// TIA Portal project "FactoryIO_assembler_analog" (V19)
// Vorlageprojekt für das Buch mit Zielsystem S7-1200

(* hardware
DEVICE "S7-1200-Station_1"  S7-1200 Station
   slot 0: "Baugruppenträger_0"  Rack  V1.0
   slot 1: "PLC_1"  CPU 1211C DC/DC/DC  6ES7 211-1AE40-0XB0  V4.1
*)

// ===== PLC "PLC_1"  CPU 1211C DC/DC/DC =====

VAR_GLOBAL   // PLC tag table "Standard-Variablentabelle"
   "lids_conveyor1" AT %A0.0 : Bool;
   "item_detected" AT %E0.0 : Bool;
   "lid_at_place" AT %E0.1 : Bool;
   "base_at_place" AT %I0.2 : Bool;
   "part_leaving" AT %I0.3 : Bool;
   "start" AT %I0.4 : Bool;
   "reset" AT %I0.5 : Bool;
   "stop" AT %I0.6 : Bool;
   "emergency_stop" AT %I0.7 : Bool;
   "auto" AT %I1.0 : Bool;
   "game_reset" AT %I1.1 : Bool;
   "x" AT %ID30 : Real;
   "z" AT %ID34 : Real;
   "stop_blade1" AT %Q0.1 : Bool;
   "lids_conveyor2" AT %Q0.2 : Bool;
   "bases_conveyor1" AT %Q0.3 : Bool;
   "stop_blade2" AT %Q0.4 : Bool;
   "bases_conveyor2" AT %Q0.5 : Bool;
   "grab" AT %Q0.6 : Bool;
   "start_light" AT %Q0.7 : Bool;
   "reset_light" AT %Q1.0 : Bool;
   "stop_light" AT %Q1.1 : Bool;
   "set_x" AT %QD30 : Real;
   "set_z" AT %QD34 : Real;
   "Counter" AT %QD38 : DInt;
   "Tag_1" AT %M0.0 : Bool;
   "Tag_2" AT %M0.1 : Bool;
   "Tag_3" AT %M0.2 : Bool;
   "item_detected_bit" AT %M0.3 : Bool;
   "grab_bit" AT %M0.4 : Bool;
   "pick_complete_bit" AT %M0.5 : Bool;
   "place_complete_bit" AT %M0.6 : Bool;
   "is_reset" AT %M0.7 : Bool;
   "home_complete_bit" AT %M1.0 : Bool;
   "Tag_4" AT %M1.1 : Bool;
END_VAR

FUNCTION "conveyor" : Void   // FC1, LAD
{ S7_Optimized_Access := 'TRUE' }
VERSION : 0.1
   VAR_TEMP   // added for the SCL form of the ladder/FBD networks
      _w1 : Bool;
      _w2 : Bool;
   END_VAR
BEGIN

REGION Network 1
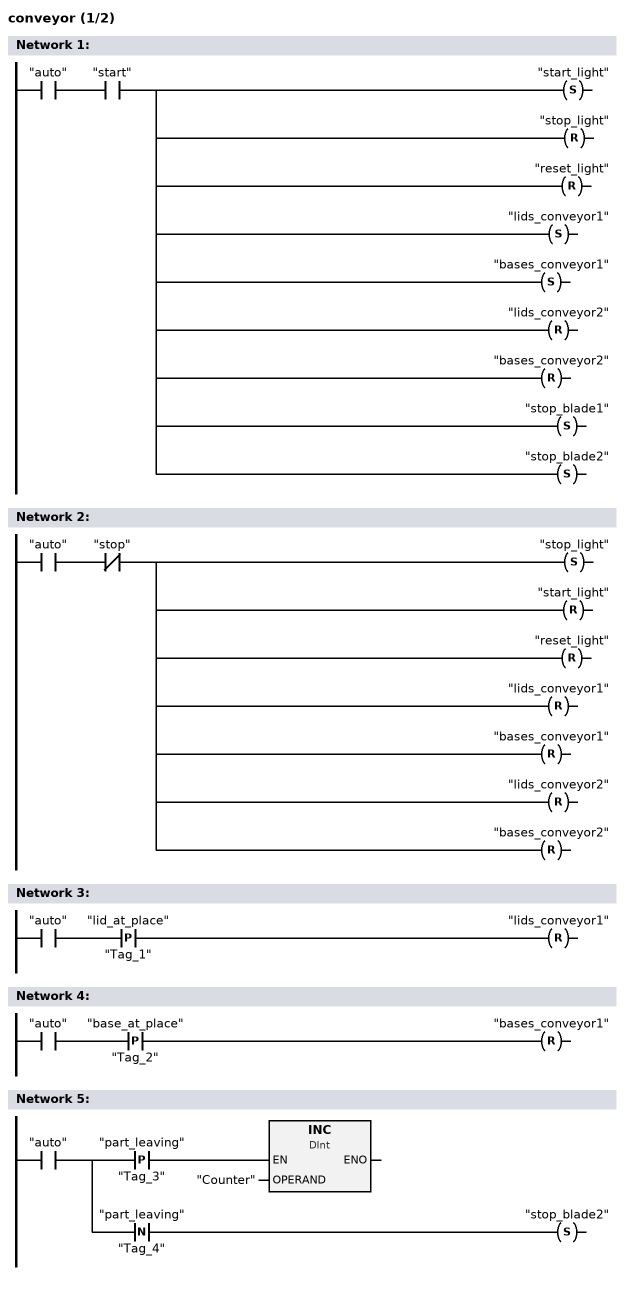
   RUNG wire#powerrail
      Contact( "auto" )
      Contact( "start" )
      wire#w1
      S_Coil( "start_light" )
   END_RUNG
   RUNG wire#w1
      R_Coil( "stop_light" )
   END_RUNG
   RUNG wire#w1
      R_Coil( "reset_light" )
   END_RUNG
   RUNG wire#w1
      S_Coil( "lids_conveyor1" )
   END_RUNG
   RUNG wire#w1
      S_Coil( "bases_conveyor1" )
   END_RUNG
   RUNG wire#w1
      R_Coil( "lids_conveyor2" )
   END_RUNG
   RUNG wire#w1
      R_Coil( "bases_conveyor2" )
   END_RUNG
   RUNG wire#w1
      S_Coil( "stop_blade1" )
   END_RUNG
   RUNG wire#w1
      S_Coil( "stop_blade2" )
   END_RUNG
   // the same network as SCL:
   IF "auto" AND "start" THEN
       "start_light" := TRUE;
       "stop_light" := FALSE;
       "reset_light" := FALSE;
       "lids_conveyor1" := TRUE;
       "bases_conveyor1" := TRUE;
       "lids_conveyor2" := FALSE;
       "bases_conveyor2" := FALSE;
       "stop_blade1" := TRUE;
       "stop_blade2" := TRUE;
   END_IF;
END_REGION

REGION Network 2
   RUNG wire#powerrail
      Contact( "auto" )
      I_Contact( "stop" )
      wire#w1
      S_Coil( "stop_light" )
   END_RUNG
   RUNG wire#w1
      R_Coil( "start_light" )
   END_RUNG
   RUNG wire#w1
      R_Coil( "reset_light" )
   END_RUNG
   RUNG wire#w1
      R_Coil( "lids_conveyor1" )
   END_RUNG
   RUNG wire#w1
      R_Coil( "bases_conveyor1" )
   END_RUNG
   RUNG wire#w1
      R_Coil( "lids_conveyor2" )
   END_RUNG
   RUNG wire#w1
      R_Coil( "bases_conveyor2" )
   END_RUNG
   // the same network as SCL:
   IF "auto" AND NOT "stop" THEN
       "stop_light" := TRUE;
       "start_light" := FALSE;
       "reset_light" := FALSE;
       "lids_conveyor1" := FALSE;
       "bases_conveyor1" := FALSE;
       "lids_conveyor2" := FALSE;
       "bases_conveyor2" := FALSE;
   END_IF;
END_REGION

REGION Network 3
   RUNG wire#powerrail
      Contact( "auto" )
      P_Contact(operand := "lid_at_place", bit := "Tag_1")
      R_Coil( "lids_conveyor1" )
   END_RUNG
   // the same network as SCL:
   #_w1 := "auto" AND "lid_at_place" AND NOT "Tag_1";   // rising edge of "lid_at_place"
   "Tag_1" := "lid_at_place";
   IF #_w1 THEN "lids_conveyor1" := FALSE; END_IF;
END_REGION

REGION Network 4
   RUNG wire#powerrail
      Contact( "auto" )
      P_Contact(operand := "base_at_place", bit := "Tag_2")
      R_Coil( "bases_conveyor1" )
   END_RUNG
   // the same network as SCL:
   #_w1 := "auto" AND "base_at_place" AND NOT "Tag_2";   // rising edge of "base_at_place"
   "Tag_2" := "base_at_place";
   IF #_w1 THEN "bases_conveyor1" := FALSE; END_IF;
END_REGION

REGION Network 5
   RUNG wire#powerrail
      Contact( "auto" )
      wire#w1
      P_Contact(operand := "part_leaving", bit := "Tag_3")
      { S7_Templates := "DestType := DInt" } Inc( "Counter" )
   END_RUNG
   RUNG wire#w1
      N_Contact(operand := "part_leaving", bit := "Tag_4")
      S_Coil( "stop_blade2" )
   END_RUNG
   // the same network as SCL:
   #_w1 := "auto" AND "part_leaving" AND NOT "Tag_3";   // rising edge of "part_leaving"
   "Tag_3" := "part_leaving";
   IF #_w1 THEN "Counter" := "Counter" + 1; END_IF;
   #_w2 := "auto" AND NOT "part_leaving" AND "Tag_4";   // falling edge of "part_leaving"
   "Tag_4" := "part_leaving";
   IF #_w2 THEN "stop_blade2" := TRUE; END_IF;
END_REGION

REGION Network 6
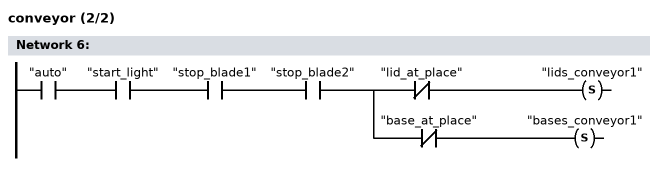
   RUNG wire#powerrail
      Contact( "auto" )
      Contact( "start_light" )
      Contact( "stop_blade1" )
      Contact( "stop_blade2" )
      wire#w1
      I_Contact( "lid_at_place" )
      S_Coil( "lids_conveyor1" )
   END_RUNG
   RUNG wire#w1
      I_Contact( "base_at_place" )
      S_Coil( "bases_conveyor1" )
   END_RUNG
   // the same network as SCL:
   #_w1 := "auto" AND "start_light" AND "stop_blade1" AND "stop_blade2";
   IF #_w1 AND NOT "lid_at_place" THEN "lids_conveyor1" := TRUE; END_IF;
   IF #_w1 AND NOT "base_at_place" THEN "bases_conveyor1" := TRUE; END_IF;
END_REGION
END_FUNCTION

FUNCTION "pick_and_place" : Void   // FC2, LAD
{ S7_Optimized_Access := 'TRUE' }
VERSION : 0.1
   VAR_TEMP
      grab_lid_x_low_limit : Real;
      grab_lid_x_high_limit : Real;
      grab_lid_z_low_limit : Real;
      grab_lid_z_high_limit : Real;
      pick_lid_z_low_limit : Real;
      pick_lid_z_high_limit : Real;
      place_lid_x_low_limit : Real;
      place_lid_x_high_limit : Real;
      place_lid_z_low_limit : Real;
      place_lid_z_high_limit : Real;
   END_VAR
   VAR CONSTANT
      grab_lid_z : Real := 9.3;
      grab_lid_x : Real := 1.2;
      offset : Real := 0.01;
      pick_lid_z : Real;
      place_lid_x : Real := 9.0;
      place_lid_z : Real := 8.95;
      home_z : Real;
      home_x : Real;
   END_VAR
   VAR_TEMP   // added for the SCL form of the ladder/FBD networks
      _w1 : Bool;
      _w2 : Bool;
   END_VAR
BEGIN

REGION Network 1 (SCL)
   // Compute limits
   // 
   #grab_lid_x_high_limit := #grab_lid_x + #offset;
   #grab_lid_x_low_limit := #grab_lid_x - #offset;

   #grab_lid_z_high_limit := #grab_lid_z + #offset;
   #grab_lid_z_low_limit := #grab_lid_z - #offset;

   #pick_lid_z_high_limit := #pick_lid_z + #offset;
   #pick_lid_z_low_limit := MAX(IN1:=0.0, IN2:=#pick_lid_z - #offset);

   #place_lid_x_high_limit:= #place_lid_x + #offset;
   #place_lid_x_low_limit:= #place_lid_x - #offset;

   #place_lid_z_high_limit:= #place_lid_z + #offset;
   #place_lid_z_low_limit:= #place_lid_z - #offset;
END_REGION

REGION Network 2: detect item
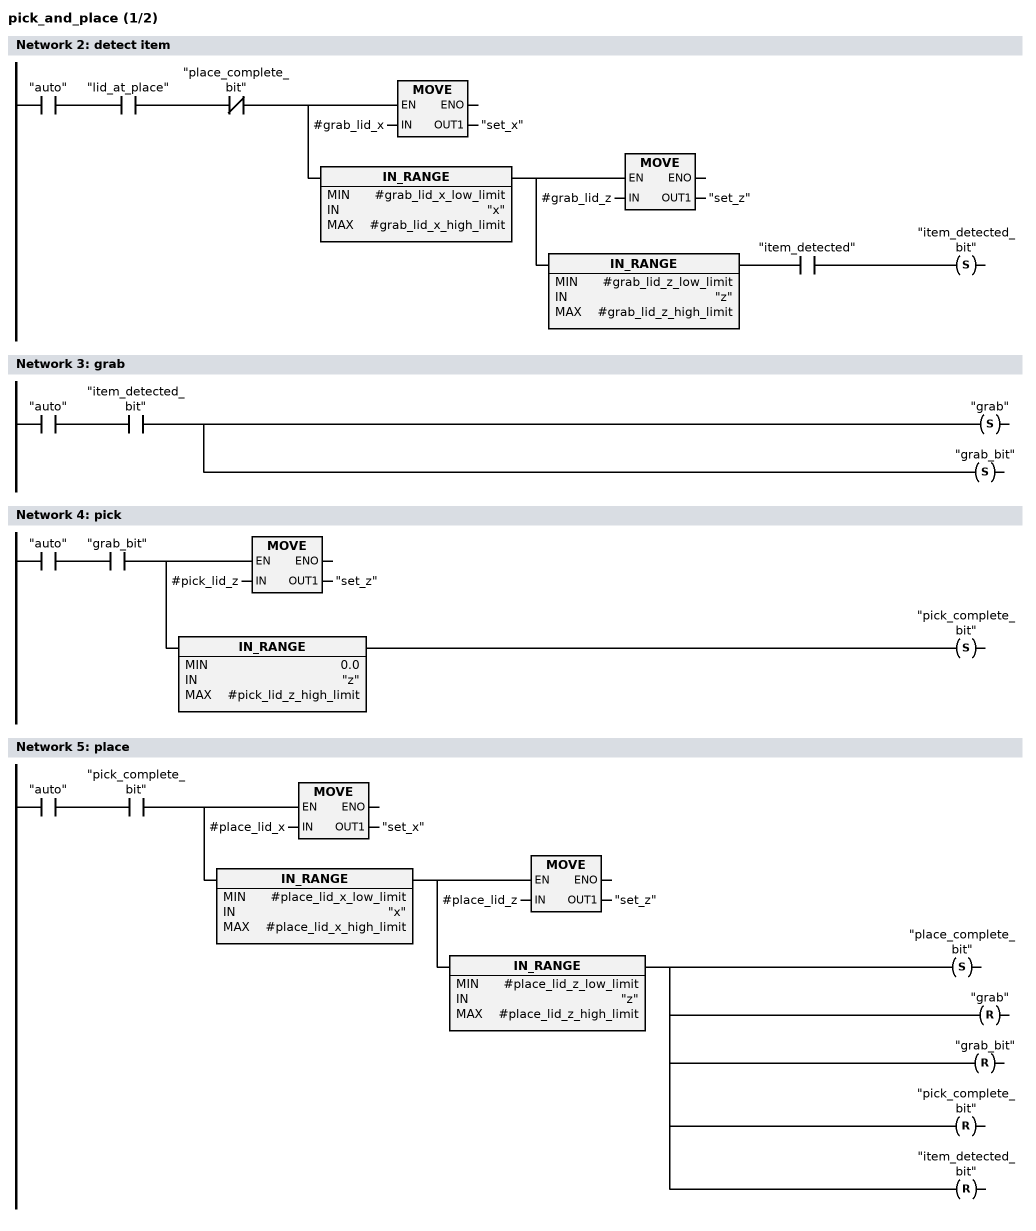
   RUNG wire#powerrail
      Contact( "auto" )
      Contact( "lid_at_place" )
      I_Contact( "place_complete_bit" )
      wire#w1
      Move(in := #grab_lid_x, out1 => "set_x")
   END_RUNG
   RUNG wire#w1
      { S7_Templates := "SrcType := Real" } InRange(min := #grab_lid_x_low_limit, in := "x", max := #grab_lid_x_high_limit)
      wire#w2
      Move(in := #grab_lid_z, out1 => "set_z")
   END_RUNG
   RUNG wire#w2
      { S7_Templates := "SrcType := Real" } InRange(min := #grab_lid_z_low_limit, in := "z", max := #grab_lid_z_high_limit)
      Contact( "item_detected" )
      S_Coil( "item_detected_bit" )
   END_RUNG
   // the same network as SCL:
   #_w1 := "auto" AND "lid_at_place" AND NOT "place_complete_bit";
   IF #_w1 THEN "set_x" := #grab_lid_x; END_IF;
   #_w2 := #_w1 AND (#grab_lid_x_low_limit <= "x") AND ("x" <= #grab_lid_x_high_limit);
   IF #_w2 THEN "set_z" := #grab_lid_z; END_IF;
   IF #_w2 AND (#grab_lid_z_low_limit <= "z") AND ("z" <= #grab_lid_z_high_limit) AND "item_detected" THEN
       "item_detected_bit" := TRUE;
   END_IF;
END_REGION

REGION Network 3: grab
   RUNG wire#powerrail
      Contact( "auto" )
      Contact( "item_detected_bit" )
      wire#w1
      S_Coil( "grab" )
   END_RUNG
   RUNG wire#w1
      S_Coil( "grab_bit" )
   END_RUNG
   // the same network as SCL:
   IF "auto" AND "item_detected_bit" THEN
       "grab" := TRUE;
       "grab_bit" := TRUE;
   END_IF;
END_REGION

REGION Network 4: pick
   RUNG wire#powerrail
      Contact( "auto" )
      Contact( "grab_bit" )
      wire#w1
      Move(in := #pick_lid_z, out1 => "set_z")
   END_RUNG
   RUNG wire#w1
      { S7_Templates := "SrcType := Real" } InRange(min := 0.0, in := "z", max := #pick_lid_z_high_limit)
      S_Coil( "pick_complete_bit" )
   END_RUNG
   // the same network as SCL:
   #_w1 := "auto" AND "grab_bit";
   IF #_w1 THEN "set_z" := #pick_lid_z; END_IF;
   IF #_w1 AND (0.0 <= "z") AND ("z" <= #pick_lid_z_high_limit) THEN "pick_complete_bit" := TRUE; END_IF;
END_REGION

REGION Network 5: place
   RUNG wire#powerrail
      Contact( "auto" )
      Contact( "pick_complete_bit" )
      wire#w1
      Move(in := #place_lid_x, out1 => "set_x")
   END_RUNG
   RUNG wire#w1
      { S7_Templates := "SrcType := Real" } InRange(min := #place_lid_x_low_limit, in := "x", max := #place_lid_x_high_limit)
      wire#w2
      Move(in := #place_lid_z, out1 => "set_z")
   END_RUNG
   RUNG wire#w2
      { S7_Templates := "SrcType := Real" } InRange(min := #place_lid_z_low_limit, in := "z", max := #place_lid_z_high_limit)
      wire#w3
      S_Coil( "place_complete_bit" )
   END_RUNG
   RUNG wire#w3
      R_Coil( "grab" )
   END_RUNG
   RUNG wire#w3
      R_Coil( "grab_bit" )
   END_RUNG
   RUNG wire#w3
      R_Coil( "pick_complete_bit" )
   END_RUNG
   RUNG wire#w3
      R_Coil( "item_detected_bit" )
   END_RUNG
   // the same network as SCL:
   #_w1 := "auto" AND "pick_complete_bit";
   IF #_w1 THEN "set_x" := #place_lid_x; END_IF;
   #_w2 := #_w1 AND (#place_lid_x_low_limit <= "x") AND ("x" <= #place_lid_x_high_limit);
   IF #_w2 THEN "set_z" := #place_lid_z; END_IF;
   IF #_w2 AND (#place_lid_z_low_limit <= "z") AND ("z" <= #place_lid_z_high_limit) THEN
       "place_complete_bit" := TRUE;
       "grab" := FALSE;
       "grab_bit" := FALSE;
       "pick_complete_bit" := FALSE;
       "item_detected_bit" := FALSE;
   END_IF;
END_REGION

REGION Network 6: home and deliver item
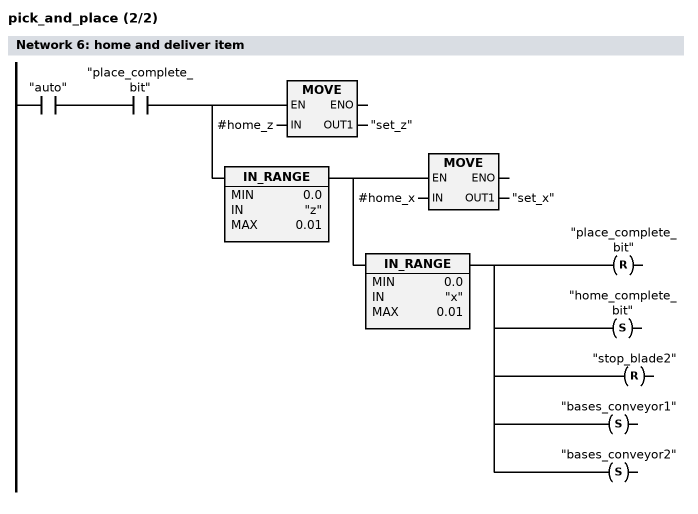
   RUNG wire#powerrail
      Contact( "auto" )
      Contact( "place_complete_bit" )
      wire#w1
      Move(in := #home_z, out1 => "set_z")
   END_RUNG
   RUNG wire#w1
      { S7_Templates := "SrcType := Real" } InRange(min := 0.0, in := "z", max := 0.01)
      wire#w2
      Move(in := #home_x, out1 => "set_x")
   END_RUNG
   RUNG wire#w2
      { S7_Templates := "SrcType := Real" } InRange(min := 0.0, in := "x", max := 0.01)
      wire#w3
      R_Coil( "place_complete_bit" )
   END_RUNG
   RUNG wire#w3
      S_Coil( "home_complete_bit" )
   END_RUNG
   RUNG wire#w3
      R_Coil( "stop_blade2" )
   END_RUNG
   RUNG wire#w3
      S_Coil( "bases_conveyor1" )
   END_RUNG
   RUNG wire#w3
      S_Coil( "bases_conveyor2" )
   END_RUNG
   // the same network as SCL:
   #_w1 := "auto" AND "place_complete_bit";
   IF #_w1 THEN "set_z" := #home_z; END_IF;
   #_w2 := #_w1 AND (0.0 <= "z") AND ("z" <= 0.01);
   IF #_w2 THEN "set_x" := #home_x; END_IF;
   IF #_w2 AND (0.0 <= "x") AND ("x" <= 0.01) THEN
       "place_complete_bit" := FALSE;
       "home_complete_bit" := TRUE;
       "stop_blade2" := FALSE;
       "bases_conveyor1" := TRUE;
       "bases_conveyor2" := TRUE;
   END_IF;
END_REGION
END_FUNCTION

FUNCTION "MHJ-PLC-Lab-Function-S71200" : Void   // FC9000, SCL
{ S7_Optimized_Access := 'TRUE' }
VERSION : 0.1
   VAR_TEMP
      rdTimeReturn : Int;
      outputTime : DTL;
      SyncVal : Byte;
      forVal : Int;
      forVal_2 : Int;
      Value : Byte;
   END_VAR
   VAR CONSTANT
      CompVal : Byte := 16#34;
      Value_01 : Byte := 16#11;
      Value_01_DW : DWord := 16#A165_D992;
      Value_02_DW : DWord := 16#58BE_4401;
   END_VAR
BEGIN

   #Value:=PEEK(area := 16#82,
        dbNumber := 0,
        byteOffset := 511);
   #Value := #Value + 1;

   POKE(area := 16#82,
        dbNumber := 0,
        byteOffset := 511,
        value := #Value);

   POKE(area:=16#81,
        dbNumber:=0,
        byteOffset:=1016,
        value:=#Value_01_DW);
   POKE(area := 16#81,
        dbNumber := 0,
        byteOffset := 1020,
        value := #Value_02_DW);

   POKE(area := 16#81,
        dbNumber := 0,
        byteOffset := 511,
        value := B#16#00);

   FOR #forVal := 0 TO 120 DO
       FOR #forVal_2:=0 TO 10 DO
           #rdTimeReturn:=RD_SYS_T(#outputTime);
           #rdTimeReturn := WR_SYS_T(#outputTime);
           #rdTimeReturn := RD_SYS_T(#outputTime);
           #rdTimeReturn := WR_SYS_T(#outputTime);
       END_FOR;
       #SyncVal:= PEEK(area := 16#81,
                      dbNumber := 0,
                      byteOffset := 511);
       IF #SyncVal = #CompVal THEN
          GOTO M_1;
       END_IF;
   END_FOR;
   RETURN;

   M_1:
   POKE(area := 16#81,
        dbNumber := 0,
        byteOffset := 511,
        value := B#16#0);
END_FUNCTION

ORGANIZATION_BLOCK "Main"   // OB1, FBD, ProgramCycle
TITLE = "Main Program Sweep (Cycle)"
{ S7_Optimized_Access := 'TRUE' }
VERSION : 0.1
   VAR_INPUT
      Initial_Call : Bool;   // Initial call of this OB
      Remanence : Bool;   // =True, if remanent data are available
   END_VAR
BEGIN

REGION Network 1: Konnektierungsbaustein für PLC-Lab
   // Im Netzwerk 1 wird der Konnektierungsbaustein für PLC-Lab aufgerufen.
   // Dieser Aufruf darf nicht entfernt werden!
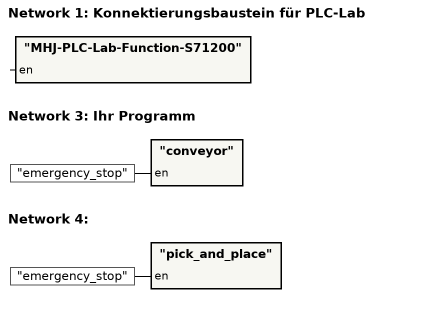
   "MHJ-PLC-Lab-Function-S71200"();
END_REGION

REGION Network 2 (SCL)
   IF "game_reset" THEN
       "start" := FALSE;
       "start_light" := FALSE;
       "reset" := FALSE;
       "reset_light" := FALSE;
       "stop" := FALSE;
       "stop_light" := FALSE;
       "bases_conveyor1" := FALSE;
       "lids_conveyor1" := FALSE;
       "grab" := FALSE;
       "grab_bit" := FALSE;
       "item_detected_bit" := FALSE;
       "pick_complete_bit" := FALSE;
       "place_complete_bit" := FALSE;
       "home_complete_bit" := FALSE;
       "set_x" := 0.0;
       "set_z" := 0.0;
       "Counter" := 0;
   END_IF;
END_REGION

REGION Network 3: Ihr Programm
   // Schreiben Sie ab Netzwerk 2 Ihr Programm
   IF "emergency_stop" THEN "conveyor"(); END_IF;
END_REGION

REGION Network 4
   IF "emergency_stop" THEN "pick_and_place"(); END_IF;
END_REGION
END_ORGANIZATION_BLOCK